// TIA Portal V19 export
VAR_GLOBAL   // PLC tag table "Default tag table"
   "EMG STOP" AT %I0.0 : Bool;
   "HOOTER RESET" AT %I0.1 : Bool;
   "PHASE FAIL" AT %I0.2 : Bool;
   "AIR PRESSURE FAIL" AT %I0.3 : Bool;
   "SYRUP MFG VESSEL BOTTOM STERROR TRIP" AT %I0.4 : Bool;
   "PREMIXING VESSEL BOTTOM STERROR TRIP" AT %I0.5 : Bool;
   "INLINE 1 HOMOGENIZER MOTOR1 TRIP" AT %I0.6 : Bool;
   "INLINE 2 HOMOGENIZER MOTOR 2 TRIP" AT %I0.7 : Bool;
   "FILTER PRESS MOTOR 1 TRIP" AT %I1.0 : Bool;
   "FILTER PRESS MOTOR 2 TRIP" AT %I1.1 : Bool;
   "VACCUM PUMP MOTOR 1 TRIP" AT %I1.2 : Bool;
   "VACCUMP PUMP MOTOR 2 TRIP" AT %I1.3 : Bool;
   "VACCUMP PUMP MOTOR 3 TRIP" AT %I1.4 : Bool;
   "VACCUMP PUMP MOTOR 4 TRIP" AT %I1.5 : Bool;
   "SUGAR VESSEL BOTTOM STERROR TRIP" AT %I1.6 : Bool;
   "BASKET FILTER MOTOR TRIP" AT %I1.7 : Bool;
   "SYRUP FLOW SWITCH" AT %I2.0 : Bool;
   "PREMIXING FLOW SWITCH" AT %I2.1 : Bool;
   "SUGAR FLOW SWITCH" AT %I2.2 : Bool;
   "INLINE 1 FLOW SWITCH" AT %I2.3 : Bool;
   "INLINE 2 FLOW SWITCH" AT %I2.4 : Bool;
   "AIR PRESSURE FAIL_2" AT %I2.5 : Bool;
   "HOOTER RESET 2" AT %I2.6 : Bool;
   SPARE_DI2 AT %I2.7 : Bool;
   SPARE_DI3 AT %I3.0 : Bool;
   SPARE_DI4 AT %I3.1 : Bool;
   SPARE_DI5 AT %I3.2 : Bool;
   SPARE_DI6 AT %I3.3 : Bool;
   SPARE_DI7 AT %I3.4 : Bool;
   SPARE_DI8 AT %I3.5 : Bool;
   SPARE_DI9 AT %I3.6 : Bool;
   EMG_STOP_2 AT %I3.7 : Bool;
   "SYRUP VESSEL TEMP SENSOR" AT %IW4 : Int;
   "PREMIXING VESSEL TEMP SENSOR" AT %IW6 : Int;
   "SUGAR VESSEL TEMP SENSOR" AT %IW8 : Int;
   "STEAM LINE_1 TEMP SENSOR" AT %IW10 : Int;
   "STEAM LINE_2 TEMP SENSOR" AT %IW12 : Int;
   "PRESSURE TRANSMITTER 1" AT %IW14 : Int;
   "PRESSURE TRANSMITTER 2" AT %IW16 : Int;
   "VACCIM TRANSMITTER 1" AT %IW18 : Int;
   "VACCIM TRANSMITTER 2" AT %IW20 : Int;
   "VACCUM TRANSMITTER 3" AT %IW22 : Int;
   "SYRUP LOAD CELL" AT %IW24 : Int;
   "PREMIXING LOAD CELL" AT %IW26 : Int;
   "SUGAR LOAD CELL" AT %IW28 : Int;
   "ULTRASONIC LEVEL SENSOR-1" AT %IW30 : Int;
   "ULTRASONIC LEVEL SENSOR-2" AT %IW32 : Int;
   "ULTRASONIC LEVEL SENSOR-3" AT %IW34 : Int;
   "SYRUP MFG VESSEL BOTTOM STERROR RUN" AT %Q0.0 : Bool;
   "PREMIXING VESSEL BOTTOM STERROR RUN" AT %Q0.1 : Bool;
   "INLINE 1 HOMOGENIZER MOTOR1 RUN" AT %Q0.2 : Bool;
   "INLINE 2 HOMOGENIZER MOTOR 2 RUN" AT %Q0.3 : Bool;
   "FILTER PRESS MOTOR 1 RUN" AT %Q0.4 : Bool;
   "FILTER PRESS MOTOR 2 RUN" AT %Q0.5 : Bool;
   "VACCUM PUMP MOTOR 1 RUN" AT %Q0.6 : Bool;
   "VACCUMP PUMP MOTOR 2 RUN" AT %Q0.7 : Bool;
   "VACCUMP PUMP MOTOR 3 RUN" AT %Q1.0 : Bool;
   "VACCUMP PUMP MOTOR 4 RUN" AT %Q1.1 : Bool;
   "SUGAR VESSEL BOTTOM STERROR RUN" AT %Q1.2 : Bool;
   "BASKET FILTER MOTOR RUN" AT %Q1.3 : Bool;
   "PBV-01" AT %Q1.4 : Bool;
   "PBV-02" AT %Q1.5 : Bool;
   "PBV-03" AT %Q1.6 : Bool;
   "PBV-04" AT %Q1.7 : Bool;
   "PBV-07" AT %Q2.0 : Bool;
   "PAV-09" AT %Q2.1 : Bool;
   "PAV-10" AT %Q2.2 : Bool;
   "PAV-11" AT %Q2.3 : Bool;
   "PAV-12" AT %Q2.4 : Bool;
   "PAV-13" AT %Q2.5 : Bool;
   "PAV-14" AT %Q2.6 : Bool;
   "PBV-15" AT %Q2.7 : Bool;
   "PBV-16" AT %Q3.0 : Bool;
   "PFBV-17" AT %Q3.1 : Bool;
   "PBV-19" AT %Q3.2 : Bool;
   "PBV-20" AT %Q3.3 : Bool;
   "PBV-21" AT %Q3.4 : Bool;
   "PBV-22" AT %Q3.5 : Bool;
   "PBV-25" AT %Q3.6 : Bool;
   "PBV-27" AT %Q3.7 : Bool;
   "PAV-28" AT %Q4.0 : Bool;
   "PAV-29" AT %Q4.1 : Bool;
   "PBV-30" AT %Q4.2 : Bool;
   "PBV-31" AT %Q4.3 : Bool;
   "PFBV-32" AT %Q4.4 : Bool;
   "PBV-36" AT %Q4.5 : Bool;
   "PBV-37" AT %Q4.6 : Bool;
   "PBV-38" AT %Q4.7 : Bool;
   "PBV-41" AT %Q5.0 : Bool;
   "PAV-50" AT %Q5.1 : Bool;
   "PAV-51" AT %Q5.2 : Bool;
   "PAV-52" AT %Q5.3 : Bool;
   "PAV-53" AT %Q5.4 : Bool;
   "PAV-54" AT %Q5.5 : Bool;
   "PAV-55" AT %Q5.6 : Bool;
   "PAV-56" AT %Q5.7 : Bool;
   "PBV-57" AT %Q6.0 : Bool;
   "PFBV-59" AT %Q6.1 : Bool;
   "PBV-79" AT %Q6.2 : Bool;
   "PBV-80" AT %Q6.3 : Bool;
   "PBV-81" AT %Q6.4 : Bool;
   "PBV-82" AT %Q6.5 : Bool;
   "PBV-83" AT %Q6.6 : Bool;
   "PBV-84" AT %Q6.7 : Bool;
   "PBV-85" AT %Q7.0 : Bool;
   "PBV-86" AT %Q7.1 : Bool;
   "PBV-87" AT %Q7.2 : Bool;
   "PBV-88" AT %Q7.3 : Bool;
   "PBV-89" AT %Q7.4 : Bool;
   "PBV-90" AT %Q7.5 : Bool;
   "PBV-91" AT %Q7.6 : Bool;
   "PBV-92" AT %Q7.7 : Bool;
   "PBV-93" AT %Q8.0 : Bool;
   "PBV-94" AT %Q8.1 : Bool;
   "PBV-95" AT %Q8.2 : Bool;
   "PBV-96" AT %Q8.3 : Bool;
   "PBV-97" AT %Q8.4 : Bool;
   "PBV-98" AT %Q8.5 : Bool;
   "PAV-99" AT %Q8.6 : Bool;
   "PBV-100" AT %Q8.7 : Bool;
   "PBV-101" AT %Q9.0 : Bool;
   "PBV-102" AT %Q9.1 : Bool;
   "PBV-103" AT %Q9.2 : Bool;
   "PBV-104" AT %Q9.3 : Bool;
   "PBV-105" AT %Q9.4 : Bool;
   "PBV-106" AT %Q9.5 : Bool;
   "PBV-107" AT %Q9.6 : Bool;
   "PBV-108" AT %Q9.7 : Bool;
   "PBV-109" AT %Q10.0 : Bool;
   "PBV-110" AT %Q10.1 : Bool;
   "PBV-111" AT %Q10.2 : Bool;
   "PBV-112" AT %Q10.3 : Bool;
   "PAV-113" AT %Q10.4 : Bool;
   "PBV-114" AT %Q10.5 : Bool;
   "PBV-115" AT %Q10.6 : Bool;
   "PBV-116" AT %Q10.7 : Bool;
   "PBV-117" AT %Q11.0 : Bool;
   "PBV-118" AT %Q11.1 : Bool;
   "PBV-119" AT %Q11.2 : Bool;
   "PBV-120" AT %Q11.3 : Bool;
   "PBV-121" AT %Q11.4 : Bool;
   "PBV-122" AT %Q11.5 : Bool;
   "PBV-123" AT %Q11.6 : Bool;
   "PBV-124" AT %Q11.7 : Bool;
   "PBV-149" AT %Q12.0 : Bool;
   "PBV-150" AT %Q12.1 : Bool;
   "PBV-151" AT %Q12.2 : Bool;
   "PBV-152" AT %Q12.3 : Bool;
   "PBV-153" AT %Q12.4 : Bool;
   "PBV-155" AT %Q12.5 : Bool;
   "PBV-156" AT %Q12.6 : Bool;
   HOOTER_1 AT %Q12.7 : Bool;
   HOOTR_2 AT %Q13.0 : Bool;
   SPARE_DO1 AT %Q13.1 : Bool;
   SPARE_DO2 AT %Q13.2 : Bool;
   SPARE_DO3 AT %Q13.3 : Bool;
   SPARE_DO4 AT %Q13.4 : Bool;
   SPARE_DO5 AT %Q13.5 : Bool;
   SPARE_DO6 AT %Q13.6 : Bool;
   SPARE_DO7 AT %Q13.7 : Bool;
   SPARE_8 AT %Q23.0 : Bool;
   SPARE_9 AT %Q23.1 : Bool;
   SPARE_10 AT %Q23.2 : Bool;
   SPARE_11 AT %Q23.3 : Bool;
   SPARE_12 AT %Q23.4 : Bool;
   SPARE_13 AT %Q23.5 : Bool;
   SPARE_14 AT %Q23.6 : Bool;
   SPARE_15 AT %Q23.7 : Bool;
   SPARE_16 AT %Q24.0 : Bool;
   SPARE_17 AT %Q24.1 : Bool;
   SPARE_18 AT %Q24.2 : Bool;
   SPARE_19 AT %Q24.3 : Bool;
   SPARE_20 AT %Q24.4 : Bool;
   SPARE_21 AT %Q24.5 : Bool;
   SPARE_22 AT %Q24.6 : Bool;
   SPARE_23 AT %Q24.7 : Bool;
   "SYRUP MFG VESSEL SPEED" AT %QW15 : Int;
   "PREMIXING VESSEL SPEED" AT %QW17 : Int;
   "SUGAR VESSEL SPEED" AT %QW19 : Int;
   "SPARE(17)" AT %QW21 : Int;
   System_Byte AT %MB1 : Byte;
   DiagStatusUpdate AT %M1.1 : Bool;
   AlwaysTRUE AT %M1.2 : Bool;
   AlwaysFALSE AT %M1.3 : Bool;
   Clock_Byte AT %MB0 : Byte;
   Clock_10Hz AT %M0.0 : Bool;
   Clock_5Hz AT %M0.1 : Bool;
   "Clock_2.5Hz" AT %M0.2 : Bool;
   Clock_2Hz AT %M0.3 : Bool;
   "Clock_1.25Hz" AT %M0.4 : Bool;
   Clock_1Hz AT %M0.5 : Bool;
   "Clock_0.625Hz" AT %M0.6 : Bool;
   "Clock_0.5Hz" AT %M0.7 : Bool;
   "Vaccup Pump2-W bit" AT %M6.0 : Bool;
   "Vaccup Pump2-S bit" AT %M6.1 : Bool;
   YY AT %M4.0 : Bool;
   "MFG LOVE CALCULATE PV" AT %MD8 : Real;
   hh1 AT %MD12 : Real;
   "MFG MOVE PV LOAD CELL" AT %MD16 : Real;
   LL AT %M2.0 : Bool;
END_VAR
